FONT_16X12:ARRAY[0..255,0..31]OF BYTE :=[
16#00,16#00,16#00,16#00,16#00,16#00,16#00,16#00,16#00,16#00,16#00,16#00,16#00,16#00,16#00,16#00,16#00,16#00,16#00,16#00,16#00,16#00,16#00,16#00,16#00,16#00,16#00,16#00,16#00,16#00,16#00,16#00,	// 16#00
16#80,16#3F,16#80,16#3F,16#C0,16#60,16#C0,16#60,16#40,16#4A,16#40,16#4A,16#40,16#43,16#40,16#43,16#40,16#43,16#40,16#43,16#40,16#4A,16#40,16#4A,16#C0,16#60,16#C0,16#60,16#80,16#3F,16#80,16#3F,	// 16#01
16#80,16#3F,16#80,16#3F,16#C0,16#7F,16#C0,16#7F,16#C0,16#75,16#C0,16#75,16#C0,16#7C,16#C0,16#7C,16#C0,16#7C,16#C0,16#7C,16#C0,16#75,16#C0,16#75,16#C0,16#7F,16#C0,16#7F,16#80,16#3F,16#80,16#3F,	// 16#02
16#00,16#0E,16#00,16#1E,16#00,16#3F,16#00,16#3F,16#80,16#3F,16#80,16#1F,16#C0,16#0F,16#C0,16#0F,16#80,16#1F,16#80,16#3F,16#00,16#3F,16#00,16#3F,16#00,16#1E,16#00,16#0E,16#00,16#00,16#00,16#00,	// 16#03
16#00,16#0C,16#00,16#0C,16#00,16#1E,16#00,16#1E,16#00,16#3F,16#00,16#3F,16#80,16#7F,16#80,16#7F,16#00,16#3F,16#00,16#3F,16#00,16#1E,16#00,16#1E,16#00,16#0C,16#00,16#0C,16#00,16#00,16#00,16#00,	// 16#04
16#00,16#0E,16#00,16#0E,16#40,16#0E,16#40,16#0E,16#40,16#3E,16#40,16#3E,16#C0,16#79,16#C0,16#79,16#C0,16#79,16#C0,16#79,16#40,16#3E,16#40,16#3E,16#40,16#0E,16#40,16#0E,16#00,16#0E,16#00,16#0E,	// 16#05
16#00,16#0C,16#00,16#0C,16#40,16#1E,16#40,16#1E,16#40,16#3E,16#40,16#3E,16#C0,16#7F,16#C0,16#7F,16#C0,16#7F,16#C0,16#7F,16#40,16#3E,16#40,16#3E,16#40,16#1E,16#40,16#1E,16#00,16#0C,16#00,16#0C,	// 16#06
16#00,16#00,16#00,16#00,16#00,16#00,16#00,16#00,16#00,16#00,16#00,16#00,16#00,16#00,16#00,16#00,16#00,16#00,16#00,16#00,16#00,16#00,16#00,16#00,16#00,16#00,16#00,16#00,16#00,16#00,16#00,16#00,	// 16#07
16#00,16#00,16#00,16#00,16#00,16#00,16#00,16#00,16#00,16#00,16#00,16#00,16#00,16#00,16#00,16#00,16#00,16#00,16#00,16#00,16#00,16#00,16#00,16#00,16#00,16#00,16#00,16#00,16#00,16#00,16#00,16#00,	// 16#08
16#00,16#00,16#00,16#00,16#00,16#00,16#00,16#00,16#00,16#00,16#00,16#00,16#00,16#00,16#00,16#00,16#00,16#00,16#00,16#00,16#00,16#00,16#00,16#00,16#00,16#00,16#00,16#00,16#00,16#00,16#00,16#00,	// 16#09
16#00,16#00,16#00,16#00,16#00,16#00,16#00,16#00,16#00,16#00,16#00,16#00,16#00,16#00,16#00,16#00,16#00,16#00,16#00,16#00,16#00,16#00,16#00,16#00,16#00,16#00,16#00,16#00,16#00,16#00,16#00,16#00,	// 16#0A
16#80,16#07,16#80,16#07,16#C0,16#0F,16#C0,16#0F,16#40,16#4C,16#40,16#4C,16#40,16#5C,16#40,16#5C,16#C0,16#77,16#C0,16#77,16#80,16#63,16#80,16#63,16#00,16#78,16#00,16#78,16#00,16#00,16#00,16#00,	// 16#0B
16#00,16#00,16#00,16#00,16#00,16#39,16#00,16#39,16#00,16#7D,16#00,16#7D,16#C0,16#47,16#C0,16#47,16#C0,16#47,16#C0,16#47,16#00,16#7D,16#00,16#7D,16#00,16#39,16#00,16#39,16#00,16#00,16#00,16#00,	// 16#0C
16#00,16#00,16#00,16#00,16#00,16#00,16#00,16#00,16#00,16#00,16#00,16#00,16#00,16#00,16#00,16#00,16#00,16#00,16#00,16#00,16#00,16#00,16#00,16#00,16#00,16#00,16#00,16#00,16#00,16#00,16#00,16#00,	// 16#0D
16#C0,16#00,16#E0,16#00,16#E0,16#7F,16#E0,16#7F,16#C0,16#7F,16#80,16#7F,16#00,16#50,16#00,16#50,16#00,16#50,16#00,16#50,16#80,16#51,16#C0,16#51,16#C0,16#7F,16#C0,16#7F,16#80,16#7F,16#00,16#7F,	// 16#0E
16#80,16#16,16#80,16#16,16#80,16#1F,16#80,16#1F,16#00,16#0F,16#00,16#0F,16#C0,16#39,16#C0,16#39,16#C0,16#39,16#C0,16#39,16#00,16#0F,16#00,16#0F,16#80,16#1F,16#80,16#1F,16#80,16#16,16#80,16#16,	// 16#0F
16#C0,16#7F,16#C0,16#7F,16#80,16#3F,16#80,16#3F,16#00,16#1F,16#00,16#1F,16#00,16#0E,16#00,16#0E,16#00,16#0E,16#00,16#0E,16#00,16#04,16#00,16#04,16#00,16#04,16#00,16#04,16#00,16#00,16#00,16#00,	// 16#10
16#00,16#04,16#00,16#04,16#00,16#04,16#00,16#04,16#00,16#0E,16#00,16#0E,16#00,16#0E,16#00,16#0E,16#00,16#1F,16#00,16#1F,16#80,16#3F,16#80,16#3F,16#C0,16#7F,16#C0,16#7F,16#00,16#00,16#00,16#00,	// 16#11
16#00,16#00,16#00,16#00,16#00,16#11,16#00,16#11,16#80,16#31,16#80,16#31,16#C0,16#7F,16#C0,16#7F,16#C0,16#7F,16#C0,16#7F,16#80,16#31,16#80,16#31,16#00,16#11,16#00,16#11,16#00,16#00,16#00,16#00,	// 16#12
16#00,16#00,16#00,16#00,16#C0,16#7C,16#C0,16#7C,16#C0,16#7C,16#C0,16#7C,16#00,16#00,16#00,16#00,16#00,16#00,16#00,16#00,16#C0,16#7C,16#C0,16#7C,16#C0,16#7C,16#C0,16#7C,16#00,16#00,16#00,16#00,	// 16#13
16#00,16#38,16#00,16#38,16#00,16#7C,16#00,16#7C,16#00,16#44,16#00,16#44,16#C0,16#7F,16#C0,16#7F,16#C0,16#7F,16#C0,16#7F,16#00,16#40,16#00,16#40,16#C0,16#7F,16#C0,16#7F,16#C0,16#7F,16#C0,16#7F,	// 16#14
16#40,16#00,16#40,16#00,16#60,16#26,16#60,16#36,16#20,16#7F,16#20,16#7F,16#20,16#59,16#20,16#49,16#20,16#49,16#A0,16#49,16#E0,16#4F,16#E0,16#4F,16#C0,16#66,16#40,16#66,16#00,16#20,16#00,16#20,	// 16#15
16#C0,16#01,16#C0,16#01,16#C0,16#01,16#C0,16#01,16#C0,16#01,16#C0,16#01,16#C0,16#01,16#C0,16#01,16#C0,16#01,16#C0,16#01,16#C0,16#01,16#C0,16#01,16#C0,16#01,16#C0,16#01,16#00,16#00,16#00,16#00,	// 16#16
16#00,16#00,16#00,16#00,16#20,16#11,16#20,16#11,16#A0,16#31,16#A0,16#31,16#E0,16#7F,16#E0,16#7F,16#E0,16#7F,16#E0,16#7F,16#A0,16#31,16#A0,16#31,16#20,16#11,16#20,16#11,16#00,16#00,16#00,16#00,	// 16#17
16#00,16#00,16#00,16#00,16#00,16#10,16#00,16#10,16#00,16#30,16#00,16#30,16#C0,16#7F,16#C0,16#7F,16#C0,16#7F,16#C0,16#7F,16#00,16#30,16#00,16#30,16#00,16#10,16#00,16#10,16#00,16#00,16#00,16#00,	// 16#18
16#00,16#00,16#00,16#00,16#00,16#01,16#00,16#01,16#80,16#01,16#80,16#01,16#C0,16#7F,16#C0,16#7F,16#C0,16#7F,16#C0,16#7F,16#80,16#01,16#80,16#01,16#00,16#01,16#00,16#01,16#00,16#00,16#00,16#00,	// 16#19
16#00,16#04,16#00,16#04,16#00,16#04,16#00,16#04,16#00,16#04,16#00,16#04,16#00,16#15,16#00,16#15,16#00,16#1F,16#00,16#1F,16#00,16#0E,16#00,16#0E,16#00,16#04,16#00,16#04,16#00,16#00,16#00,16#00,	// 16#1A
16#00,16#04,16#00,16#04,16#00,16#0E,16#00,16#0E,16#00,16#1F,16#00,16#1F,16#00,16#15,16#00,16#15,16#00,16#04,16#00,16#04,16#00,16#04,16#00,16#04,16#00,16#04,16#00,16#04,16#00,16#00,16#00,16#00,	// 16#1B
16#00,16#0F,16#00,16#0F,16#00,16#0F,16#00,16#0F,16#00,16#01,16#00,16#01,16#00,16#01,16#00,16#01,16#00,16#01,16#00,16#01,16#00,16#01,16#00,16#01,16#00,16#01,16#00,16#01,16#00,16#00,16#00,16#00,	// 16#1C
16#00,16#04,16#00,16#04,16#00,16#0E,16#00,16#0E,16#00,16#1F,16#00,16#1F,16#00,16#04,16#00,16#04,16#00,16#04,16#00,16#04,16#00,16#1F,16#00,16#1F,16#00,16#0E,16#00,16#0E,16#00,16#04,16#00,16#04,	// 16#1D
16#C0,16#00,16#C0,16#01,16#C0,16#03,16#C0,16#07,16#C0,16#0F,16#C0,16#1F,16#C0,16#3F,16#C0,16#3F,16#C0,16#1F,16#C0,16#0F,16#C0,16#07,16#C0,16#03,16#C0,16#01,16#C0,16#00,16#00,16#00,16#00,16#00,	// 16#1E
16#00,16#30,16#00,16#38,16#00,16#3C,16#00,16#3E,16#00,16#3F,16#80,16#3F,16#C0,16#3F,16#C0,16#3F,16#80,16#3F,16#00,16#3F,16#00,16#3E,16#00,16#3C,16#00,16#38,16#00,16#30,16#00,16#00,16#00,16#00,	// 16#1F
16#00,16#00,16#00,16#00,16#00,16#00,16#00,16#00,16#00,16#00,16#00,16#00,16#00,16#00,16#00,16#00,16#00,16#00,16#00,16#00,16#00,16#00,16#00,16#00,16#00,16#00,16#00,16#00,16#00,16#00,16#00,16#00,	// 16#20
16#00,16#00,16#00,16#00,16#00,16#10,16#00,16#38,16#C0,16#7E,16#C0,16#7E,16#C0,16#7E,16#C0,16#7E,16#00,16#38,16#00,16#10,16#00,16#00,16#00,16#00,16#00,16#00,16#00,16#00,16#00,16#00,16#00,16#00,	// 16#21
16#00,16#00,16#00,16#00,16#00,16#60,16#00,16#70,16#00,16#78,16#00,16#78,16#00,16#00,16#00,16#00,16#00,16#00,16#00,16#00,16#00,16#78,16#00,16#78,16#00,16#70,16#00,16#60,16#00,16#00,16#00,16#00,	// 16#22
16#00,16#11,16#00,16#11,16#C0,16#7F,16#C0,16#7F,16#C0,16#7F,16#C0,16#7F,16#00,16#11,16#00,16#11,16#C0,16#7F,16#C0,16#7F,16#C0,16#7F,16#C0,16#7F,16#00,16#11,16#00,16#11,16#00,16#00,16#00,16#00,	// 16#23
16#80,16#18,16#80,16#18,16#80,16#3C,16#80,16#3C,16#E0,16#E4,16#E0,16#E4,16#E0,16#E4,16#E0,16#E4,16#80,16#27,16#80,16#27,16#00,16#23,16#00,16#23,16#00,16#00,16#00,16#00,16#00,16#00,16#00,16#00,	// 16#24
16#C0,16#18,16#C0,16#18,16#80,16#19,16#80,16#19,16#00,16#03,16#00,16#03,16#00,16#06,16#00,16#06,16#C0,16#0C,16#C0,16#0C,16#C0,16#18,16#C0,16#18,16#00,16#00,16#00,16#00,16#00,16#00,16#00,16#00,	// 16#25
16#80,16#37,16#80,16#37,16#C0,16#7F,16#C0,16#7F,16#40,16#4C,16#40,16#4C,16#C0,16#7C,16#C0,16#7E,16#80,16#37,16#80,16#37,16#C0,16#03,16#C0,16#02,16#40,16#06,16#40,16#06,16#00,16#00,16#00,16#00,	// 16#26
16#00,16#00,16#00,16#00,16#00,16#08,16#00,16#08,16#00,16#78,16#00,16#78,16#00,16#70,16#00,16#60,16#00,16#00,16#00,16#00,16#00,16#00,16#00,16#00,16#00,16#00,16#00,16#00,16#00,16#00,16#00,16#00,	// 16#27
16#00,16#00,16#00,16#00,16#00,16#1F,16#00,16#1F,16#80,16#3F,16#80,16#3F,16#C0,16#60,16#C0,16#60,16#40,16#40,16#40,16#40,16#00,16#00,16#00,16#00,16#00,16#00,16#00,16#00,16#00,16#00,16#00,16#00,	// 16#28
16#00,16#00,16#00,16#00,16#00,16#00,16#00,16#00,16#40,16#40,16#40,16#40,16#C0,16#60,16#C0,16#60,16#80,16#3F,16#80,16#3F,16#00,16#1F,16#00,16#1F,16#00,16#00,16#00,16#00,16#00,16#00,16#00,16#00,	// 16#29
16#00,16#04,16#00,16#04,16#00,16#15,16#00,16#15,16#00,16#1F,16#00,16#1F,16#00,16#0E,16#00,16#0E,16#00,16#0E,16#00,16#0E,16#00,16#1F,16#00,16#1F,16#00,16#15,16#00,16#15,16#00,16#04,16#00,16#04,	// 16#2A
16#00,16#00,16#00,16#00,16#00,16#04,16#00,16#04,16#00,16#04,16#00,16#04,16#00,16#1F,16#00,16#1F,16#00,16#1F,16#00,16#1F,16#00,16#04,16#00,16#04,16#00,16#04,16#00,16#04,16#00,16#00,16#00,16#00,	// 16#2B
16#00,16#00,16#00,16#00,16#20,16#00,16#20,16#00,16#E0,16#00,16#E0,16#00,16#C0,16#00,16#C0,16#00,16#C0,16#00,16#80,16#00,16#00,16#00,16#00,16#00,16#00,16#00,16#00,16#00,16#00,16#00,16#00,16#00,	// 16#2C
16#00,16#04,16#00,16#04,16#00,16#04,16#00,16#04,16#00,16#04,16#00,16#04,16#00,16#04,16#00,16#04,16#00,16#04,16#00,16#04,16#00,16#04,16#00,16#04,16#00,16#04,16#00,16#04,16#00,16#00,16#00,16#00,	// 16#2D
16#00,16#00,16#00,16#00,16#00,16#00,16#00,16#00,16#C0,16#00,16#C0,16#00,16#C0,16#00,16#C0,16#00,16#C0,16#00,16#C0,16#00,16#00,16#00,16#00,16#00,16#00,16#00,16#00,16#00,16#00,16#00,16#00,16#00,	// 16#2E
16#C0,16#00,16#C0,16#00,16#80,16#01,16#80,16#01,16#00,16#03,16#00,16#03,16#00,16#06,16#00,16#06,16#00,16#0C,16#00,16#0C,16#00,16#18,16#00,16#18,16#00,16#30,16#00,16#30,16#00,16#00,16#00,16#00,	// 16#2F
16#80,16#3F,16#80,16#3F,16#C0,16#7F,16#C0,16#7F,16#C0,16#41,16#40,16#43,16#40,16#46,16#40,16#4C,16#40,16#58,16#40,16#70,16#C0,16#7F,16#C0,16#7F,16#80,16#3F,16#80,16#3F,16#00,16#00,16#00,16#00,	// 16#30
16#40,16#10,16#40,16#10,16#40,16#10,16#40,16#10,16#C0,16#3F,16#C0,16#3F,16#C0,16#7F,16#C0,16#7F,16#40,16#00,16#40,16#00,16#40,16#00,16#40,16#00,16#00,16#00,16#00,16#00,16#00,16#00,16#00,16#00,	// 16#31
16#C0,16#30,16#C0,16#30,16#C0,16#71,16#C0,16#71,16#40,16#43,16#40,16#43,16#40,16#46,16#40,16#46,16#C0,16#7C,16#C0,16#7C,16#C0,16#38,16#C0,16#38,16#00,16#00,16#00,16#00,16#00,16#00,16#00,16#00,	// 16#32
16#80,16#20,16#80,16#20,16#C0,16#60,16#C0,16#60,16#40,16#44,16#40,16#44,16#40,16#44,16#40,16#44,16#C0,16#7F,16#C0,16#7F,16#80,16#3B,16#80,16#3B,16#00,16#00,16#00,16#00,16#00,16#00,16#00,16#00,	// 16#33
16#00,16#06,16#00,16#06,16#00,16#0E,16#00,16#0E,16#00,16#1A,16#00,16#1A,16#40,16#32,16#40,16#32,16#C0,16#7F,16#C0,16#7F,16#C0,16#7F,16#C0,16#7F,16#40,16#02,16#40,16#02,16#00,16#00,16#00,16#00,	// 16#34
16#80,16#7C,16#80,16#7C,16#C0,16#7C,16#C0,16#7C,16#40,16#44,16#40,16#44,16#40,16#44,16#40,16#44,16#C0,16#47,16#C0,16#47,16#80,16#43,16#80,16#43,16#00,16#00,16#00,16#00,16#00,16#00,16#00,16#00,	// 16#35
16#80,16#1F,16#80,16#1F,16#C0,16#3F,16#C0,16#3F,16#40,16#64,16#40,16#64,16#40,16#44,16#40,16#44,16#C0,16#47,16#C0,16#47,16#80,16#03,16#80,16#03,16#00,16#00,16#00,16#00,16#00,16#00,16#00,16#00,	// 16#36
16#00,16#70,16#00,16#70,16#00,16#70,16#00,16#70,16#C0,16#41,16#C0,16#41,16#C0,16#43,16#C0,16#43,16#00,16#46,16#00,16#46,16#00,16#7C,16#00,16#7C,16#00,16#78,16#00,16#78,16#00,16#00,16#00,16#00,	// 16#37
16#80,16#3B,16#80,16#3B,16#C0,16#7F,16#C0,16#7F,16#40,16#44,16#40,16#44,16#40,16#44,16#40,16#44,16#C0,16#7F,16#C0,16#7F,16#80,16#3B,16#80,16#3B,16#00,16#00,16#00,16#00,16#00,16#00,16#00,16#00,	// 16#38
16#00,16#38,16#00,16#38,16#40,16#7C,16#40,16#7C,16#C0,16#44,16#C0,16#44,16#C0,16#47,16#C0,16#47,16#00,16#7F,16#00,16#7F,16#00,16#3C,16#00,16#3C,16#00,16#00,16#00,16#00,16#00,16#00,16#00,16#00,	// 16#39
16#00,16#00,16#00,16#00,16#00,16#00,16#00,16#00,16#80,16#19,16#80,16#19,16#80,16#19,16#80,16#19,16#80,16#19,16#80,16#19,16#00,16#00,16#00,16#00,16#00,16#00,16#00,16#00,16#00,16#00,16#00,16#00,	// 16#3A
16#00,16#00,16#00,16#00,16#00,16#00,16#00,16#00,16#A0,16#19,16#A0,16#19,16#E0,16#19,16#E0,16#19,16#C0,16#19,16#C0,16#19,16#00,16#00,16#00,16#00,16#00,16#00,16#00,16#00,16#00,16#00,16#00,16#00,	// 16#3B
16#00,16#04,16#00,16#04,16#00,16#0E,16#00,16#0E,16#00,16#1B,16#00,16#1B,16#80,16#31,16#80,16#31,16#C0,16#60,16#C0,16#60,16#40,16#40,16#40,16#40,16#00,16#00,16#00,16#00,16#00,16#00,16#00,16#00,	// 16#3C
16#00,16#00,16#00,16#00,16#00,16#0A,16#00,16#0A,16#00,16#0A,16#00,16#0A,16#00,16#0A,16#00,16#0A,16#00,16#0A,16#00,16#0A,16#00,16#0A,16#00,16#0A,16#00,16#0A,16#00,16#0A,16#00,16#00,16#00,16#00,	// 16#3D
16#00,16#00,16#00,16#00,16#40,16#40,16#40,16#40,16#C0,16#60,16#C0,16#60,16#80,16#31,16#80,16#31,16#00,16#1B,16#00,16#1B,16#00,16#0E,16#00,16#0E,16#00,16#04,16#00,16#04,16#00,16#00,16#00,16#00,	// 16#3E
16#00,16#20,16#00,16#20,16#00,16#60,16#00,16#60,16#C0,16#46,16#C0,16#46,16#C0,16#4E,16#C0,16#4E,16#00,16#78,16#00,16#78,16#00,16#30,16#00,16#30,16#00,16#00,16#00,16#00,16#00,16#00,16#00,16#00,	// 16#3F
16#80,16#3F,16#80,16#3F,16#C0,16#7F,16#C0,16#7F,16#40,16#40,16#40,16#40,16#40,16#4E,16#40,16#4E,16#40,16#4A,16#40,16#4A,16#40,16#7A,16#40,16#7E,16#00,16#3E,16#00,16#3E,16#00,16#00,16#00,16#00,	// 16#40
16#C0,16#1F,16#C0,16#1F,16#C0,16#3F,16#C0,16#3F,16#00,16#62,16#00,16#62,16#00,16#62,16#00,16#62,16#C0,16#3F,16#C0,16#3F,16#C0,16#1F,16#C0,16#1F,16#00,16#00,16#00,16#00,16#00,16#00,16#00,16#00,	// 16#41
16#40,16#40,16#40,16#40,16#C0,16#7F,16#C0,16#7F,16#C0,16#7F,16#C0,16#7F,16#40,16#44,16#40,16#44,16#40,16#44,16#40,16#44,16#C0,16#7F,16#C0,16#7F,16#80,16#3B,16#80,16#3B,16#00,16#00,16#00,16#00,	// 16#42
16#00,16#1F,16#00,16#1F,16#80,16#3F,16#80,16#3F,16#C0,16#60,16#C0,16#60,16#40,16#40,16#40,16#40,16#40,16#40,16#40,16#40,16#C0,16#71,16#C0,16#71,16#80,16#31,16#80,16#31,16#00,16#00,16#00,16#00,	// 16#43
16#40,16#40,16#40,16#40,16#C0,16#7F,16#C0,16#7F,16#C0,16#7F,16#C0,16#7F,16#40,16#40,16#40,16#40,16#C0,16#60,16#C0,16#60,16#80,16#3F,16#80,16#3F,16#00,16#1F,16#00,16#1F,16#00,16#00,16#00,16#00,	// 16#44
16#40,16#40,16#40,16#40,16#C0,16#7F,16#C0,16#7F,16#C0,16#7F,16#C0,16#7F,16#40,16#44,16#40,16#44,16#40,16#44,16#40,16#44,16#40,16#4E,16#40,16#4E,16#C0,16#60,16#C0,16#60,16#00,16#00,16#00,16#00,	// 16#45
16#40,16#40,16#40,16#40,16#C0,16#7F,16#C0,16#7F,16#C0,16#7F,16#C0,16#7F,16#40,16#44,16#40,16#44,16#00,16#44,16#00,16#44,16#00,16#6E,16#00,16#6E,16#00,16#70,16#00,16#70,16#00,16#00,16#00,16#00,	// 16#46
16#00,16#1F,16#00,16#1F,16#80,16#3F,16#80,16#3F,16#C0,16#60,16#C0,16#60,16#40,16#40,16#40,16#40,16#40,16#42,16#40,16#42,16#C0,16#73,16#C0,16#73,16#C0,16#33,16#C0,16#33,16#00,16#00,16#00,16#00,	// 16#47
16#C0,16#7F,16#C0,16#7F,16#C0,16#7F,16#C0,16#7F,16#00,16#04,16#00,16#04,16#00,16#04,16#00,16#04,16#C0,16#7F,16#C0,16#7F,16#C0,16#7F,16#C0,16#7F,16#00,16#00,16#00,16#00,16#00,16#00,16#00,16#00,	// 16#48
16#00,16#00,16#00,16#00,16#40,16#40,16#40,16#40,16#C0,16#7F,16#C0,16#7F,16#C0,16#7F,16#C0,16#7F,16#40,16#40,16#40,16#40,16#00,16#00,16#00,16#00,16#00,16#00,16#00,16#00,16#00,16#00,16#00,16#00,	// 16#49
16#80,16#03,16#80,16#03,16#C0,16#03,16#C0,16#03,16#40,16#00,16#40,16#00,16#40,16#40,16#40,16#40,16#C0,16#7F,16#C0,16#7F,16#80,16#7F,16#80,16#7F,16#00,16#40,16#00,16#40,16#00,16#00,16#00,16#00,	// 16#4A
16#40,16#40,16#40,16#40,16#C0,16#7F,16#C0,16#7F,16#C0,16#7F,16#C0,16#7F,16#00,16#04,16#00,16#04,16#00,16#0E,16#00,16#1F,16#C0,16#7B,16#C0,16#71,16#C0,16#60,16#C0,16#60,16#00,16#00,16#00,16#00,	// 16#4B
16#40,16#40,16#40,16#40,16#C0,16#7F,16#C0,16#7F,16#C0,16#7F,16#C0,16#7F,16#40,16#40,16#40,16#40,16#40,16#00,16#40,16#00,16#C0,16#01,16#C0,16#01,16#C0,16#03,16#C0,16#03,16#00,16#00,16#00,16#00,	// 16#4C
16#C0,16#7F,16#C0,16#7F,16#C0,16#7F,16#C0,16#7F,16#00,16#38,16#00,16#38,16#00,16#1C,16#00,16#1C,16#00,16#38,16#00,16#38,16#C0,16#7F,16#C0,16#7F,16#C0,16#7F,16#C0,16#7F,16#00,16#00,16#00,16#00,	// 16#4D
16#C0,16#7F,16#C0,16#7F,16#C0,16#7F,16#C0,16#7F,16#00,16#1C,16#00,16#1C,16#00,16#0E,16#00,16#0E,16#00,16#07,16#00,16#07,16#C0,16#7F,16#C0,16#7F,16#C0,16#7F,16#C0,16#7F,16#00,16#00,16#00,16#00,	// 16#4E
16#00,16#1F,16#00,16#1F,16#80,16#3F,16#80,16#3F,16#C0,16#71,16#C0,16#60,16#40,16#40,16#40,16#40,16#C0,16#60,16#C0,16#71,16#80,16#3F,16#80,16#3F,16#00,16#1F,16#00,16#1F,16#00,16#00,16#00,16#00,	// 16#4F
16#40,16#40,16#40,16#40,16#C0,16#7F,16#C0,16#7F,16#C0,16#7F,16#C0,16#7F,16#40,16#44,16#40,16#44,16#00,16#44,16#00,16#44,16#00,16#7C,16#00,16#7C,16#00,16#38,16#00,16#38,16#00,16#00,16#00,16#00,	// 16#50
16#00,16#1F,16#00,16#1F,16#80,16#3F,16#80,16#3F,16#80,16#60,16#80,16#60,16#A0,16#40,16#A0,16#43,16#E0,16#63,16#E0,16#61,16#E0,16#3F,16#E0,16#3F,16#20,16#1F,16#20,16#1F,16#00,16#00,16#00,16#00,	// 16#51
16#40,16#40,16#40,16#40,16#C0,16#7F,16#C0,16#7F,16#C0,16#7F,16#C0,16#7F,16#00,16#44,16#00,16#44,16#00,16#46,16#00,16#46,16#C0,16#7F,16#C0,16#7F,16#C0,16#39,16#C0,16#39,16#00,16#00,16#00,16#00,	// 16#52
16#80,16#39,16#80,16#39,16#C0,16#7D,16#C0,16#7D,16#40,16#44,16#40,16#44,16#40,16#46,16#40,16#46,16#C0,16#73,16#C0,16#73,16#80,16#31,16#80,16#31,16#00,16#00,16#00,16#00,16#00,16#00,16#00,16#00,	// 16#53
16#00,16#60,16#00,16#60,16#40,16#40,16#40,16#40,16#C0,16#7F,16#C0,16#7F,16#C0,16#7F,16#C0,16#7F,16#40,16#40,16#40,16#40,16#00,16#60,16#00,16#60,16#00,16#00,16#00,16#00,16#00,16#00,16#00,16#00,	// 16#54
16#80,16#7F,16#80,16#7F,16#C0,16#7F,16#C0,16#7F,16#40,16#00,16#40,16#00,16#40,16#00,16#40,16#00,16#C0,16#7F,16#C0,16#7F,16#80,16#7F,16#80,16#7F,16#00,16#00,16#00,16#00,16#00,16#00,16#00,16#00,	// 16#55
16#00,16#7F,16#00,16#7F,16#80,16#7F,16#80,16#7F,16#C0,16#00,16#C0,16#00,16#C0,16#00,16#C0,16#00,16#80,16#7F,16#80,16#7F,16#00,16#7F,16#00,16#7F,16#00,16#00,16#00,16#00,16#00,16#00,16#00,16#00,	// 16#56
16#00,16#7E,16#00,16#7F,16#C0,16#7F,16#C0,16#7F,16#C0,16#01,16#C0,16#03,16#00,16#07,16#00,16#07,16#C0,16#03,16#C0,16#01,16#C0,16#7F,16#C0,16#7F,16#00,16#7F,16#00,16#7E,16#00,16#00,16#00,16#00,	// 16#57
16#C0,16#71,16#C0,16#71,16#C0,16#7B,16#C0,16#7B,16#00,16#0E,16#00,16#0E,16#00,16#0E,16#00,16#0E,16#C0,16#7B,16#C0,16#7B,16#C0,16#71,16#C0,16#71,16#00,16#00,16#00,16#00,16#00,16#00,16#00,16#00,	// 16#58
16#00,16#78,16#00,16#78,16#40,16#7C,16#40,16#7C,16#C0,16#07,16#C0,16#07,16#C0,16#07,16#C0,16#07,16#40,16#7C,16#40,16#7C,16#00,16#78,16#00,16#78,16#00,16#00,16#00,16#00,16#00,16#00,16#00,16#00,	// 16#59
16#C0,16#70,16#C0,16#71,16#C0,16#61,16#C0,16#63,16#40,16#47,16#40,16#46,16#40,16#4C,16#40,16#5C,16#40,16#58,16#40,16#58,16#C0,16#70,16#C0,16#70,16#C0,16#61,16#C0,16#61,16#00,16#00,16#00,16#00,	// 16#5A
16#00,16#00,16#00,16#00,16#00,16#00,16#00,16#00,16#C0,16#7F,16#C0,16#7F,16#C0,16#7F,16#C0,16#7F,16#40,16#40,16#40,16#40,16#40,16#40,16#40,16#40,16#00,16#00,16#00,16#00,16#00,16#00,16#00,16#00,	// 16#5B
16#00,16#30,16#00,16#30,16#00,16#18,16#00,16#18,16#00,16#0C,16#00,16#0C,16#00,16#06,16#00,16#06,16#00,16#03,16#00,16#03,16#80,16#01,16#80,16#01,16#C0,16#00,16#C0,16#00,16#00,16#00,16#00,16#00,	// 16#5C
16#00,16#00,16#00,16#00,16#00,16#00,16#00,16#00,16#40,16#40,16#40,16#40,16#40,16#40,16#40,16#40,16#C0,16#7F,16#C0,16#7F,16#C0,16#7F,16#C0,16#7F,16#00,16#00,16#00,16#00,16#00,16#00,16#00,16#00,	// 16#5D
16#00,16#10,16#00,16#10,16#00,16#30,16#00,16#30,16#00,16#60,16#00,16#60,16#00,16#C0,16#00,16#C0,16#00,16#60,16#00,16#60,16#00,16#30,16#00,16#30,16#00,16#10,16#00,16#10,16#00,16#00,16#00,16#00,	// 16#5E
16#20,16#00,16#20,16#00,16#20,16#00,16#20,16#00,16#20,16#00,16#20,16#00,16#20,16#00,16#20,16#00,16#20,16#00,16#20,16#00,16#20,16#00,16#20,16#00,16#20,16#00,16#20,16#00,16#20,16#00,16#20,16#00,	// 16#5F
16#00,16#00,16#00,16#00,16#00,16#00,16#00,16#00,16#00,16#C0,16#00,16#C0,16#00,16#E0,16#00,16#E0,16#00,16#20,16#00,16#20,16#00,16#00,16#00,16#00,16#00,16#00,16#00,16#00,16#00,16#00,16#00,16#00,	// 16#60
16#80,16#01,16#80,16#01,16#C0,16#0B,16#C0,16#0B,16#40,16#0A,16#40,16#0A,16#40,16#0A,16#40,16#0A,16#C0,16#0F,16#80,16#0F,16#80,16#07,16#C0,16#07,16#40,16#00,16#40,16#00,16#00,16#00,16#00,16#00,	// 16#61
16#40,16#40,16#40,16#40,16#C0,16#7F,16#80,16#7F,16#80,16#7F,16#C0,16#7F,16#40,16#08,16#40,16#08,16#40,16#08,16#40,16#08,16#C0,16#0F,16#C0,16#0F,16#80,16#07,16#80,16#07,16#00,16#00,16#00,16#00,	// 16#62
16#80,16#07,16#80,16#07,16#C0,16#0F,16#C0,16#0F,16#40,16#08,16#40,16#08,16#40,16#08,16#40,16#08,16#C0,16#0C,16#C0,16#0C,16#80,16#04,16#80,16#04,16#00,16#00,16#00,16#00,16#00,16#00,16#00,16#00,	// 16#63
16#80,16#07,16#80,16#07,16#C0,16#0F,16#C0,16#0F,16#40,16#08,16#40,16#08,16#40,16#48,16#40,16#48,16#C0,16#7F,16#80,16#7F,16#80,16#7F,16#C0,16#7F,16#40,16#00,16#40,16#00,16#00,16#00,16#00,16#00,	// 16#64
16#80,16#07,16#80,16#07,16#C0,16#0F,16#C0,16#0F,16#40,16#0A,16#40,16#0A,16#40,16#0A,16#40,16#0A,16#C0,16#0E,16#C0,16#0E,16#80,16#06,16#80,16#06,16#00,16#00,16#00,16#00,16#00,16#00,16#00,16#00,	// 16#65
16#40,16#04,16#40,16#04,16#C0,16#3F,16#C0,16#3F,16#C0,16#7F,16#C0,16#7F,16#40,16#44,16#40,16#44,16#00,16#64,16#00,16#64,16#00,16#20,16#00,16#20,16#00,16#00,16#00,16#00,16#00,16#00,16#00,16#00,	// 16#66
16#20,16#07,16#20,16#07,16#B0,16#0F,16#B0,16#0F,16#90,16#08,16#90,16#08,16#90,16#08,16#90,16#08,16#F0,16#0F,16#F0,16#07,16#E0,16#07,16#E0,16#0F,16#00,16#08,16#00,16#08,16#00,16#00,16#00,16#00,	// 16#67
16#40,16#40,16#40,16#40,16#C0,16#7F,16#C0,16#7F,16#C0,16#7F,16#C0,16#7F,16#00,16#04,16#00,16#04,16#00,16#08,16#00,16#08,16#C0,16#0F,16#C0,16#0F,16#C0,16#07,16#C0,16#07,16#00,16#00,16#00,16#00,	// 16#68
16#00,16#00,16#00,16#00,16#40,16#08,16#40,16#08,16#40,16#08,16#40,16#08,16#C0,16#6F,16#C0,16#6F,16#C0,16#6F,16#C0,16#6F,16#40,16#00,16#40,16#00,16#40,16#00,16#40,16#00,16#00,16#00,16#00,16#00,	// 16#69
16#60,16#00,16#60,16#00,16#70,16#00,16#70,16#00,16#10,16#08,16#10,16#08,16#10,16#08,16#10,16#08,16#F0,16#6F,16#F0,16#6F,16#E0,16#6F,16#E0,16#6F,16#00,16#00,16#00,16#00,16#00,16#00,16#00,16#00,	// 16#6A
16#40,16#40,16#40,16#40,16#C0,16#7F,16#C0,16#7F,16#C0,16#7F,16#C0,16#7F,16#00,16#02,16#00,16#02,16#00,16#07,16#00,16#07,16#C0,16#0D,16#C0,16#0D,16#C0,16#08,16#C0,16#08,16#00,16#00,16#00,16#00,	// 16#6B
16#00,16#00,16#00,16#00,16#40,16#40,16#40,16#40,16#40,16#40,16#40,16#40,16#C0,16#7F,16#C0,16#7F,16#C0,16#7F,16#C0,16#7F,16#40,16#00,16#40,16#00,16#40,16#00,16#40,16#00,16#00,16#00,16#00,16#00,	// 16#6C
16#C0,16#0F,16#C0,16#0F,16#C0,16#0F,16#C0,16#0F,16#00,16#08,16#00,16#08,16#80,16#0F,16#80,16#0F,16#00,16#08,16#00,16#08,16#C0,16#0F,16#C0,16#0F,16#C0,16#07,16#C0,16#07,16#00,16#00,16#00,16#00,	// 16#6D
16#C0,16#0F,16#C0,16#0F,16#C0,16#0F,16#C0,16#0F,16#00,16#08,16#00,16#08,16#00,16#08,16#00,16#08,16#C0,16#0F,16#C0,16#0F,16#C0,16#07,16#C0,16#07,16#00,16#00,16#00,16#00,16#00,16#00,16#00,16#00,	// 16#6E
16#80,16#07,16#80,16#07,16#C0,16#0F,16#C0,16#0F,16#40,16#08,16#40,16#08,16#40,16#08,16#40,16#08,16#C0,16#0F,16#C0,16#0F,16#80,16#07,16#80,16#07,16#00,16#00,16#00,16#00,16#00,16#00,16#00,16#00,	// 16#6F
16#10,16#08,16#10,16#08,16#F0,16#0F,16#F0,16#07,16#F0,16#07,16#F0,16#0F,16#50,16#08,16#50,16#08,16#40,16#08,16#40,16#08,16#C0,16#0F,16#C0,16#0F,16#80,16#07,16#80,16#07,16#00,16#00,16#00,16#00,	// 16#70
16#80,16#07,16#80,16#07,16#C0,16#0F,16#C0,16#0F,16#40,16#08,16#40,16#08,16#50,16#08,16#50,16#08,16#F0,16#0F,16#F0,16#07,16#F0,16#07,16#F0,16#0F,16#10,16#08,16#10,16#08,16#00,16#00,16#00,16#00,	// 16#71
16#40,16#08,16#40,16#08,16#C0,16#0F,16#C0,16#0F,16#C0,16#0F,16#C0,16#0F,16#40,16#02,16#40,16#06,16#00,16#0C,16#00,16#0C,16#00,16#0E,16#00,16#0E,16#00,16#06,16#00,16#06,16#00,16#00,16#00,16#00,	// 16#72
16#80,16#04,16#80,16#04,16#C0,16#0E,16#C0,16#0E,16#40,16#0A,16#40,16#0B,16#40,16#0B,16#40,16#09,16#C0,16#0D,16#C0,16#0D,16#80,16#04,16#80,16#04,16#00,16#00,16#00,16#00,16#00,16#00,16#00,16#00,	// 16#73
16#00,16#08,16#00,16#08,16#80,16#1F,16#80,16#1F,16#C0,16#3F,16#C0,16#3F,16#40,16#08,16#40,16#08,16#C0,16#08,16#C0,16#08,16#80,16#08,16#80,16#08,16#00,16#00,16#00,16#00,16#00,16#00,16#00,16#00,	// 16#74
16#80,16#0F,16#80,16#0F,16#C0,16#0F,16#C0,16#0F,16#40,16#00,16#40,16#00,16#40,16#00,16#40,16#00,16#80,16#0F,16#80,16#0F,16#C0,16#0F,16#C0,16#0F,16#40,16#00,16#40,16#00,16#00,16#00,16#00,16#00,	// 16#75
16#00,16#0F,16#00,16#0F,16#80,16#0F,16#80,16#0F,16#C0,16#00,16#C0,16#00,16#C0,16#00,16#C0,16#00,16#80,16#0F,16#80,16#0F,16#00,16#0F,16#00,16#0F,16#00,16#00,16#00,16#00,16#00,16#00,16#00,16#00,	// 16#76
16#00,16#0F,16#00,16#0F,16#C0,16#0F,16#C0,16#0F,16#C0,16#00,16#C0,16#00,16#00,16#03,16#00,16#03,16#C0,16#00,16#C0,16#00,16#C0,16#0F,16#C0,16#0F,16#00,16#0F,16#00,16#0F,16#00,16#00,16#00,16#00,	// 16#77
16#40,16#08,16#40,16#08,16#C0,16#0C,16#C0,16#0C,16#80,16#07,16#80,16#07,16#00,16#03,16#00,16#03,16#80,16#07,16#80,16#07,16#C0,16#0C,16#C0,16#0C,16#40,16#08,16#40,16#08,16#00,16#00,16#00,16#00,	// 16#78
16#10,16#00,16#10,16#00,16#10,16#0F,16#10,16#0F,16#90,16#0F,16#90,16#0F,16#B0,16#00,16#B0,16#00,16#E0,16#00,16#E0,16#00,16#C0,16#0F,16#C0,16#0F,16#00,16#0F,16#00,16#0F,16#00,16#00,16#00,16#00,	// 16#79
16#C0,16#0C,16#C0,16#0C,16#C0,16#09,16#C0,16#09,16#40,16#09,16#40,16#0B,16#40,16#0B,16#40,16#0A,16#40,16#0E,16#40,16#0E,16#C0,16#0C,16#C0,16#0C,16#00,16#00,16#00,16#00,16#00,16#00,16#00,16#00,	// 16#7A
16#00,16#04,16#00,16#04,16#00,16#0E,16#00,16#0E,16#80,16#3B,16#80,16#3B,16#C0,16#71,16#C0,16#71,16#40,16#40,16#40,16#40,16#40,16#40,16#40,16#40,16#00,16#00,16#00,16#00,16#00,16#00,16#00,16#00,	// 16#7B
16#00,16#00,16#00,16#00,16#00,16#00,16#00,16#00,16#00,16#00,16#00,16#00,16#C0,16#7B,16#C0,16#7B,16#C0,16#7B,16#C0,16#7B,16#00,16#00,16#00,16#00,16#00,16#00,16#00,16#00,16#00,16#00,16#00,16#00,	// 16#7C
16#40,16#40,16#40,16#40,16#40,16#40,16#40,16#40,16#C0,16#71,16#C0,16#71,16#80,16#3B,16#80,16#3B,16#00,16#0E,16#00,16#0E,16#00,16#04,16#00,16#04,16#00,16#00,16#00,16#00,16#00,16#00,16#00,16#00,	// 16#7D
16#00,16#30,16#00,16#30,16#00,16#70,16#00,16#60,16#00,16#40,16#00,16#40,16#00,16#60,16#00,16#60,16#00,16#30,16#00,16#30,16#00,16#10,16#00,16#10,16#00,16#30,16#00,16#70,16#00,16#60,16#00,16#40,	// 16#7E
16#80,16#03,16#80,16#03,16#80,16#07,16#80,16#07,16#80,16#0C,16#80,16#0C,16#80,16#18,16#80,16#18,16#80,16#0C,16#80,16#0C,16#80,16#07,16#80,16#07,16#80,16#03,16#80,16#03,16#00,16#00,16#00,16#00,	// 16#7F
16#80,16#3F,16#90,16#3F,16#D0,16#7F,16#D0,16#7F,16#70,16#40,16#70,16#40,16#70,16#40,16#60,16#40,16#C0,16#71,16#C0,16#71,16#80,16#31,16#80,16#31,16#00,16#00,16#00,16#00,16#00,16#00,16#00,16#00,	// 16#80
16#80,16#6F,16#80,16#6F,16#C0,16#6F,16#C0,16#6F,16#40,16#00,16#40,16#00,16#40,16#00,16#40,16#00,16#C0,16#6F,16#80,16#6F,16#80,16#6F,16#C0,16#6F,16#40,16#00,16#40,16#00,16#00,16#00,16#00,16#00,	// 16#81
16#80,16#07,16#80,16#07,16#C0,16#0F,16#C0,16#0F,16#40,16#2A,16#40,16#2A,16#40,16#6A,16#40,16#6A,16#C0,16#CE,16#C0,16#CE,16#80,16#86,16#80,16#86,16#00,16#00,16#00,16#00,16#00,16#00,16#00,16#00,	// 16#82
16#80,16#21,16#80,16#21,16#C0,16#6B,16#C0,16#6B,16#40,16#CA,16#40,16#CA,16#40,16#CA,16#40,16#CA,16#C0,16#6F,16#80,16#6F,16#80,16#27,16#C0,16#27,16#40,16#00,16#40,16#00,16#00,16#00,16#00,16#00,	// 16#83
16#80,16#61,16#80,16#61,16#C0,16#6B,16#C0,16#6B,16#40,16#0A,16#40,16#0A,16#40,16#0A,16#40,16#0A,16#C0,16#6F,16#80,16#6F,16#80,16#67,16#C0,16#67,16#40,16#00,16#40,16#00,16#00,16#00,16#00,16#00,	// 16#84
16#80,16#81,16#80,16#81,16#C0,16#CB,16#C0,16#CB,16#40,16#6A,16#40,16#6A,16#40,16#2A,16#40,16#2A,16#C0,16#0F,16#80,16#0F,16#80,16#07,16#C0,16#07,16#40,16#00,16#40,16#00,16#00,16#00,16#00,16#00,	// 16#85
16#80,16#09,16#80,16#09,16#C0,16#6B,16#C0,16#6B,16#40,16#FA,16#40,16#FA,16#40,16#9A,16#40,16#9A,16#C0,16#FF,16#80,16#FF,16#80,16#67,16#C0,16#67,16#40,16#00,16#40,16#00,16#00,16#00,16#00,16#00,	// 16#86
16#80,16#07,16#90,16#07,16#D0,16#0F,16#D0,16#0F,16#70,16#08,16#70,16#08,16#70,16#08,16#60,16#08,16#C0,16#0C,16#C0,16#0C,16#80,16#04,16#80,16#04,16#00,16#00,16#00,16#00,16#00,16#00,16#00,16#00,	// 16#87
16#80,16#27,16#80,16#27,16#C0,16#6F,16#C0,16#6F,16#40,16#CA,16#40,16#CA,16#40,16#CA,16#40,16#CA,16#40,16#6E,16#40,16#6E,16#40,16#26,16#40,16#26,16#00,16#00,16#00,16#00,16#00,16#00,16#00,16#00,	// 16#88
16#80,16#67,16#80,16#67,16#C0,16#6F,16#C0,16#6F,16#40,16#0A,16#40,16#0A,16#40,16#0A,16#40,16#0A,16#40,16#6E,16#40,16#6E,16#40,16#66,16#40,16#66,16#00,16#00,16#00,16#00,16#00,16#00,16#00,16#00,	// 16#89
16#80,16#87,16#80,16#87,16#C0,16#CF,16#C0,16#CF,16#40,16#6A,16#40,16#6A,16#40,16#2A,16#40,16#2A,16#40,16#0E,16#40,16#0E,16#40,16#06,16#40,16#06,16#00,16#00,16#00,16#00,16#00,16#00,16#00,16#00,	// 16#8A
16#00,16#00,16#00,16#00,16#40,16#68,16#40,16#68,16#40,16#68,16#40,16#68,16#C0,16#0F,16#C0,16#0F,16#C0,16#6F,16#C0,16#6F,16#40,16#60,16#40,16#60,16#40,16#00,16#40,16#00,16#00,16#00,16#00,16#00,	// 16#8B
16#00,16#00,16#00,16#00,16#40,16#28,16#40,16#28,16#40,16#68,16#40,16#68,16#C0,16#CF,16#C0,16#CF,16#C0,16#6F,16#C0,16#6F,16#40,16#20,16#40,16#20,16#40,16#00,16#40,16#00,16#00,16#00,16#00,16#00,	// 16#8C
16#00,16#00,16#00,16#00,16#40,16#88,16#40,16#88,16#40,16#C8,16#40,16#C8,16#C0,16#6F,16#C0,16#6F,16#C0,16#2F,16#C0,16#2F,16#40,16#00,16#40,16#00,16#40,16#00,16#40,16#00,16#00,16#00,16#00,16#00,	// 16#8D
16#C0,16#47,16#C0,16#47,16#C0,16#4F,16#C0,16#4F,16#00,16#19,16#00,16#19,16#00,16#19,16#00,16#19,16#C0,16#4F,16#C0,16#4F,16#C0,16#47,16#C0,16#47,16#00,16#00,16#00,16#00,16#00,16#00,16#00,16#00,	// 16#8E
16#C0,16#67,16#C0,16#67,16#C0,16#FF,16#C0,16#FF,16#00,16#99,16#00,16#99,16#00,16#99,16#00,16#99,16#C0,16#FF,16#C0,16#FF,16#C0,16#67,16#C0,16#67,16#00,16#00,16#00,16#00,16#00,16#00,16#00,16#00,	// 16#8F
16#C0,16#1F,16#C0,16#1F,16#C0,16#1F,16#C0,16#1F,16#40,16#32,16#40,16#32,16#40,16#72,16#40,16#72,16#40,16#D2,16#40,16#D2,16#C0,16#98,16#C0,16#98,16#00,16#00,16#00,16#00,16#00,16#00,16#00,16#00,	// 16#90
16#C0,16#01,16#C0,16#09,16#C0,16#0B,16#C0,16#0B,16#40,16#0A,16#40,16#0A,16#C0,16#0A,16#80,16#0F,16#80,16#0F,16#C0,16#0F,16#C0,16#0A,16#40,16#0A,16#40,16#0A,16#40,16#0E,16#40,16#06,16#40,16#06,	// 16#91
16#C0,16#1F,16#C0,16#1F,16#C0,16#3F,16#C0,16#3F,16#00,16#64,16#00,16#64,16#C0,16#7F,16#C0,16#7F,16#C0,16#7F,16#C0,16#7F,16#40,16#44,16#40,16#44,16#40,16#44,16#40,16#44,16#00,16#00,16#00,16#00,	// 16#92
16#80,16#27,16#80,16#27,16#C0,16#6F,16#C0,16#6F,16#40,16#C8,16#40,16#C8,16#40,16#C8,16#40,16#C8,16#C0,16#6F,16#C0,16#6F,16#80,16#27,16#80,16#27,16#00,16#00,16#00,16#00,16#00,16#00,16#00,16#00,	// 16#93
16#80,16#67,16#80,16#67,16#C0,16#6F,16#C0,16#6F,16#40,16#08,16#40,16#08,16#40,16#08,16#40,16#08,16#C0,16#6F,16#C0,16#6F,16#80,16#67,16#80,16#67,16#00,16#00,16#00,16#00,16#00,16#00,16#00,16#00,	// 16#94
16#80,16#87,16#80,16#87,16#C0,16#CF,16#C0,16#CF,16#40,16#68,16#40,16#68,16#40,16#28,16#40,16#28,16#C0,16#0F,16#C0,16#0F,16#80,16#07,16#80,16#07,16#00,16#00,16#00,16#00,16#00,16#00,16#00,16#00,	// 16#95
16#80,16#2F,16#80,16#2F,16#C0,16#6F,16#C0,16#6F,16#40,16#C0,16#40,16#C0,16#40,16#C0,16#40,16#C0,16#C0,16#6F,16#80,16#6F,16#80,16#2F,16#C0,16#2F,16#40,16#00,16#40,16#00,16#00,16#00,16#00,16#00,	// 16#96
16#80,16#8F,16#80,16#8F,16#C0,16#CF,16#C0,16#CF,16#40,16#60,16#40,16#60,16#40,16#20,16#40,16#20,16#C0,16#0F,16#80,16#0F,16#80,16#0F,16#C0,16#0F,16#40,16#00,16#40,16#00,16#00,16#00,16#00,16#00,	// 16#97
16#10,16#00,16#10,16#00,16#10,16#6F,16#10,16#6F,16#90,16#6F,16#90,16#6F,16#B0,16#00,16#B0,16#00,16#E0,16#00,16#E0,16#00,16#C0,16#6F,16#C0,16#6F,16#00,16#6F,16#00,16#6F,16#00,16#00,16#00,16#00,	// 16#98
16#80,16#4F,16#80,16#4F,16#C0,16#5F,16#C0,16#1F,16#40,16#10,16#40,16#10,16#40,16#10,16#40,16#10,16#C0,16#1F,16#C0,16#5F,16#80,16#4F,16#80,16#4F,16#00,16#00,16#00,16#00,16#00,16#00,16#00,16#00,	// 16#99
16#80,16#BF,16#80,16#BF,16#C0,16#BF,16#C0,16#BF,16#40,16#00,16#40,16#00,16#40,16#00,16#40,16#00,16#C0,16#BF,16#C0,16#BF,16#80,16#BF,16#80,16#BF,16#00,16#00,16#00,16#00,16#00,16#00,16#00,16#00,	// 16#9A
16#80,16#07,16#80,16#07,16#C0,16#0F,16#C0,16#0F,16#C0,16#09,16#40,16#0B,16#40,16#0E,16#40,16#0C,16#C0,16#0F,16#C0,16#07,16#80,16#07,16#80,16#07,16#00,16#00,16#00,16#00,16#00,16#00,16#00,16#00,	// 16#9B
16#C0,16#04,16#C0,16#04,16#C0,16#7F,16#C0,16#7F,16#40,16#FF,16#40,16#FF,16#40,16#84,16#40,16#84,16#40,16#84,16#40,16#84,16#40,16#C4,16#40,16#C4,16#40,16#40,16#40,16#40,16#00,16#00,16#00,16#00,	// 16#9C
16#00,16#1F,16#40,16#1F,16#C0,16#3F,16#80,16#3F,16#C0,16#71,16#C0,16#63,16#40,16#46,16#40,16#4C,16#C0,16#78,16#C0,16#71,16#80,16#3F,16#80,16#7F,16#00,16#5F,16#00,16#1F,16#00,16#00,16#00,16#00,	// 16#9D
16#40,16#08,16#C0,16#0C,16#C0,16#0C,16#80,16#04,16#80,16#07,16#00,16#03,16#00,16#03,16#00,16#03,16#80,16#07,16#80,16#04,16#C0,16#0C,16#C0,16#0C,16#40,16#08,16#00,16#00,16#00,16#00,16#00,16#00,	// 16#9E
16#80,16#00,16#80,16#00,16#C0,16#08,16#C0,16#08,16#40,16#08,16#40,16#08,16#C0,16#7F,16#C0,16#7F,16#80,16#FF,16#80,16#FF,16#00,16#88,16#00,16#88,16#00,16#C8,16#00,16#C8,16#00,16#40,16#00,16#40,	// 16#9F
16#80,16#01,16#80,16#01,16#C0,16#0B,16#C0,16#0B,16#40,16#2A,16#40,16#2A,16#40,16#6A,16#40,16#6A,16#C0,16#CF,16#80,16#CF,16#80,16#87,16#C0,16#87,16#40,16#00,16#40,16#00,16#00,16#00,16#00,16#00,	// 16#A0
16#00,16#00,16#00,16#00,16#40,16#08,16#40,16#08,16#40,16#28,16#40,16#28,16#C0,16#6F,16#C0,16#6F,16#C0,16#CF,16#C0,16#CF,16#40,16#80,16#40,16#80,16#40,16#00,16#40,16#00,16#00,16#00,16#00,16#00,	// 16#A1
16#80,16#07,16#80,16#07,16#C0,16#0F,16#C0,16#0F,16#40,16#28,16#40,16#28,16#40,16#68,16#40,16#68,16#C0,16#CF,16#C0,16#CF,16#80,16#87,16#80,16#87,16#00,16#00,16#00,16#00,16#00,16#00,16#00,16#00,	// 16#A2
16#80,16#0F,16#80,16#0F,16#C0,16#0F,16#C0,16#0F,16#40,16#20,16#40,16#20,16#40,16#60,16#40,16#60,16#C0,16#CF,16#80,16#CF,16#80,16#8F,16#C0,16#8F,16#40,16#00,16#40,16#00,16#00,16#00,16#00,16#00,	// 16#A3
16#C0,16#2F,16#C0,16#2F,16#C0,16#6F,16#C0,16#6F,16#00,16#48,16#00,16#48,16#00,16#68,16#00,16#68,16#C0,16#2F,16#C0,16#2F,16#C0,16#67,16#C0,16#67,16#00,16#40,16#00,16#40,16#00,16#00,16#00,16#00,	// 16#A4
16#C0,16#5F,16#C0,16#5F,16#C0,16#DF,16#C0,16#DF,16#00,16#8C,16#00,16#8C,16#00,16#C6,16#00,16#C6,16#00,16#43,16#00,16#43,16#C0,16#DF,16#C0,16#DF,16#C0,16#9F,16#C0,16#9F,16#00,16#00,16#00,16#00,	// 16#A5
16#00,16#32,16#00,16#32,16#00,16#7A,16#00,16#7A,16#00,16#4A,16#00,16#4A,16#00,16#4A,16#00,16#4A,16#00,16#7A,16#00,16#72,16#00,16#72,16#00,16#7A,16#00,16#0A,16#00,16#0A,16#00,16#00,16#00,16#00,	// 16#A6
16#00,16#32,16#00,16#32,16#00,16#7A,16#00,16#7A,16#00,16#4A,16#00,16#4A,16#00,16#4A,16#00,16#4A,16#00,16#7A,16#00,16#7A,16#00,16#32,16#00,16#32,16#00,16#02,16#00,16#02,16#00,16#00,16#00,16#00,	// 16#A7
16#80,16#03,16#80,16#03,16#C0,16#07,16#C0,16#07,16#40,16#6C,16#40,16#6C,16#40,16#68,16#40,16#68,16#C0,16#00,16#C0,16#00,16#80,16#00,16#80,16#00,16#00,16#00,16#00,16#00,16#00,16#00,16#00,16#00,	// 16#A8
16#00,16#1F,16#80,16#3F,16#C0,16#60,16#40,16#5F,16#40,16#5F,16#40,16#54,16#40,16#5E,16#40,16#5B,16#40,16#41,16#C0,16#60,16#80,16#3F,16#00,16#1F,16#00,16#00,16#00,16#00,16#00,16#00,16#00,16#00,	// 16#A9
16#00,16#04,16#00,16#04,16#00,16#04,16#00,16#04,16#00,16#04,16#00,16#04,16#00,16#04,16#00,16#04,16#80,16#07,16#80,16#07,16#80,16#07,16#80,16#07,16#00,16#00,16#00,16#00,16#00,16#00,16#00,16#00,	// 16#AA
16#80,16#21,16#80,16#21,16#00,16#7B,16#00,16#7B,16#00,16#7E,16#00,16#7E,16#20,16#0C,16#20,16#0D,16#60,16#1B,16#60,16#1A,16#E0,16#32,16#E0,16#32,16#A0,16#63,16#A0,16#63,16#20,16#01,16#20,16#01,	// 16#AB
16#80,16#21,16#80,16#21,16#00,16#7B,16#00,16#7B,16#C0,16#7E,16#C0,16#7E,16#C0,16#0D,16#C0,16#0D,16#40,16#1B,16#40,16#1B,16#40,16#36,16#40,16#36,16#E0,16#67,16#E0,16#67,16#E0,16#47,16#E0,16#47,	// 16#AC
16#00,16#00,16#00,16#00,16#80,16#03,16#80,16#03,16#C0,16#6F,16#C0,16#6F,16#C0,16#6F,16#C0,16#6F,16#80,16#03,16#80,16#03,16#00,16#00,16#00,16#00,16#00,16#00,16#00,16#00,16#00,16#00,16#00,16#00,	// 16#AD
16#00,16#03,16#00,16#03,16#80,16#07,16#80,16#07,16#C0,16#0C,16#C0,16#0C,16#40,16#08,16#40,16#08,16#00,16#03,16#00,16#03,16#80,16#07,16#80,16#07,16#C0,16#0C,16#C0,16#0C,16#40,16#08,16#40,16#08,	// 16#AE
16#40,16#08,16#40,16#08,16#C0,16#0C,16#C0,16#0C,16#80,16#07,16#80,16#07,16#00,16#03,16#00,16#03,16#40,16#08,16#40,16#08,16#C0,16#0C,16#C0,16#0C,16#80,16#07,16#80,16#07,16#00,16#03,16#00,16#03,	// 16#AF
16#20,16#49,16#20,16#49,16#90,16#24,16#90,16#24,16#40,16#92,16#40,16#92,16#20,16#49,16#20,16#49,16#90,16#24,16#90,16#24,16#40,16#92,16#40,16#92,16#20,16#49,16#20,16#49,16#90,16#24,16#90,16#24,	// 16#B0
16#50,16#55,16#50,16#55,16#A0,16#AA,16#A0,16#AA,16#50,16#55,16#50,16#55,16#A0,16#AA,16#A0,16#AA,16#50,16#55,16#50,16#55,16#A0,16#AA,16#A0,16#AA,16#50,16#55,16#50,16#55,16#A0,16#AA,16#A0,16#AA,	// 16#B1
16#B0,16#6D,16#B0,16#6D,16#60,16#DB,16#60,16#DB,16#D0,16#B6,16#D0,16#B6,16#B0,16#6D,16#B0,16#6D,16#60,16#DB,16#60,16#DB,16#D0,16#B6,16#D0,16#B6,16#B0,16#6D,16#B0,16#6D,16#60,16#DB,16#60,16#DB,	// 16#B2
16#00,16#00,16#00,16#00,16#00,16#00,16#00,16#00,16#00,16#00,16#00,16#00,16#F0,16#FF,16#F0,16#FF,16#F0,16#FF,16#F0,16#FF,16#00,16#00,16#00,16#00,16#00,16#00,16#00,16#00,16#00,16#00,16#00,16#00,	// 16#B3
16#00,16#00,16#00,16#00,16#00,16#04,16#00,16#04,16#00,16#04,16#00,16#04,16#F0,16#FF,16#F0,16#FF,16#F0,16#FF,16#F0,16#FF,16#00,16#00,16#00,16#00,16#00,16#00,16#00,16#00,16#00,16#00,16#00,16#00,	// 16#B4
16#C0,16#07,16#C0,16#0F,16#C0,16#0F,16#C0,16#1F,16#00,16#51,16#00,16#51,16#00,16#D1,16#00,16#D1,16#C0,16#9F,16#C0,16#8F,16#C0,16#0F,16#C0,16#07,16#00,16#00,16#00,16#00,16#00,16#00,16#00,16#00,	// 16#B5
16#C0,16#07,16#C0,16#0F,16#C0,16#4F,16#C0,16#5F,16#00,16#D1,16#00,16#91,16#00,16#91,16#00,16#D1,16#C0,16#5F,16#C0,16#4F,16#C0,16#0F,16#C0,16#07,16#00,16#00,16#00,16#00,16#00,16#00,16#00,16#00,	// 16#B6
16#C0,16#07,16#C0,16#0F,16#C0,16#8F,16#C0,16#9F,16#00,16#D1,16#00,16#D1,16#00,16#51,16#00,16#51,16#C0,16#1F,16#C0,16#0F,16#C0,16#0F,16#C0,16#07,16#00,16#00,16#00,16#00,16#00,16#00,16#00,16#00,	// 16#B7
16#00,16#1F,16#80,16#3F,16#C0,16#60,16#40,16#4E,16#40,16#5F,16#40,16#51,16#40,16#51,16#40,16#51,16#40,16#40,16#C0,16#60,16#80,16#3F,16#00,16#1F,16#00,16#00,16#00,16#00,16#00,16#00,16#00,16#00,	// 16#B8
16#00,16#09,16#00,16#09,16#F0,16#F9,16#F0,16#F9,16#F0,16#F9,16#F0,16#F9,16#00,16#00,16#00,16#00,16#00,16#00,16#00,16#00,16#F0,16#FF,16#F0,16#FF,16#F0,16#FF,16#F0,16#FF,16#00,16#00,16#00,16#00,	// 16#B9
16#00,16#00,16#00,16#00,16#F0,16#FF,16#F0,16#FF,16#F0,16#FF,16#F0,16#FF,16#00,16#00,16#00,16#00,16#00,16#00,16#00,16#00,16#F0,16#FF,16#F0,16#FF,16#F0,16#FF,16#F0,16#FF,16#00,16#00,16#00,16#00,	// 16#BA
16#00,16#09,16#00,16#09,16#F0,16#09,16#F0,16#09,16#F0,16#09,16#F0,16#09,16#00,16#08,16#00,16#08,16#00,16#08,16#00,16#08,16#F0,16#0F,16#F0,16#0F,16#F0,16#0F,16#F0,16#0F,16#00,16#00,16#00,16#00,	// 16#BB
16#00,16#09,16#00,16#09,16#00,16#F9,16#00,16#F9,16#00,16#F9,16#00,16#F9,16#00,16#01,16#00,16#01,16#00,16#01,16#00,16#01,16#00,16#FF,16#00,16#FF,16#00,16#FF,16#00,16#FF,16#00,16#00,16#00,16#00,	// 16#BC
16#00,16#04,16#00,16#04,16#00,16#FC,16#00,16#FC,16#00,16#FC,16#00,16#FC,16#00,16#04,16#00,16#04,16#00,16#04,16#00,16#04,16#00,16#FC,16#00,16#FC,16#00,16#FC,16#00,16#FC,16#00,16#00,16#00,16#00,	// 16#BD
16#00,16#0F,16#00,16#0F,16#80,16#1F,16#80,16#1F,16#E0,16#70,16#E0,16#70,16#E0,16#70,16#E0,16#70,16#80,16#19,16#80,16#19,16#00,16#09,16#00,16#09,16#00,16#00,16#00,16#00,16#00,16#00,16#00,16#00,	// 16#BE
16#00,16#F5,16#00,16#F5,16#00,16#FD,16#00,16#FD,16#C0,16#0F,16#C0,16#0F,16#C0,16#0F,16#C0,16#0F,16#00,16#FD,16#00,16#FD,16#00,16#F5,16#00,16#F5,16#00,16#00,16#00,16#00,16#00,16#00,16#00,16#00,	// 16#BF
16#00,16#00,16#00,16#00,16#00,16#00,16#00,16#00,16#00,16#00,16#00,16#00,16#00,16#FC,16#00,16#FC,16#00,16#FC,16#00,16#FC,16#00,16#04,16#00,16#04,16#00,16#04,16#00,16#04,16#00,16#04,16#00,16#04,	// 16#C0
16#00,16#04,16#00,16#04,16#00,16#04,16#00,16#04,16#00,16#04,16#00,16#04,16#00,16#FC,16#00,16#FC,16#00,16#FC,16#00,16#FC,16#00,16#04,16#00,16#04,16#00,16#04,16#00,16#04,16#00,16#04,16#00,16#04,	// 16#C1
16#00,16#04,16#00,16#04,16#00,16#04,16#00,16#04,16#00,16#04,16#00,16#04,16#F0,16#07,16#F0,16#07,16#F0,16#07,16#F0,16#07,16#00,16#04,16#00,16#04,16#00,16#04,16#00,16#04,16#00,16#04,16#00,16#04,	// 16#C2
16#00,16#00,16#00,16#00,16#00,16#00,16#00,16#00,16#00,16#00,16#00,16#00,16#F0,16#FF,16#F0,16#FF,16#F0,16#FF,16#F0,16#FF,16#00,16#04,16#00,16#04,16#00,16#04,16#00,16#04,16#00,16#04,16#00,16#04,	// 16#C3
16#00,16#04,16#00,16#04,16#00,16#04,16#00,16#04,16#00,16#04,16#00,16#04,16#00,16#04,16#00,16#04,16#00,16#04,16#00,16#04,16#00,16#04,16#00,16#04,16#00,16#04,16#00,16#04,16#00,16#04,16#00,16#04,	// 16#C4
16#00,16#04,16#00,16#04,16#00,16#04,16#00,16#04,16#00,16#04,16#00,16#04,16#F0,16#FF,16#F0,16#FF,16#F0,16#FF,16#F0,16#FF,16#00,16#04,16#00,16#04,16#00,16#04,16#00,16#04,16#00,16#04,16#00,16#04,	// 16#C5
16#80,16#21,16#80,16#21,16#C0,16#6B,16#C0,16#6B,16#40,16#4A,16#40,16#4A,16#40,16#6A,16#40,16#6A,16#C0,16#2F,16#80,16#2F,16#80,16#67,16#C0,16#67,16#40,16#40,16#40,16#40,16#00,16#00,16#00,16#00,	// 16#C6
16#C0,16#47,16#C0,16#4F,16#C0,16#CF,16#C0,16#DF,16#00,16#91,16#00,16#D1,16#00,16#D1,16#00,16#51,16#C0,16#DF,16#C0,16#CF,16#C0,16#8F,16#C0,16#87,16#00,16#00,16#00,16#00,16#00,16#00,16#00,16#00,	// 16#C7
16#00,16#00,16#00,16#00,16#00,16#FF,16#00,16#FF,16#00,16#FF,16#00,16#FF,16#00,16#01,16#00,16#01,16#00,16#01,16#00,16#01,16#00,16#F9,16#00,16#F9,16#00,16#F9,16#00,16#F9,16#00,16#09,16#00,16#09,	// 16#C8
16#00,16#00,16#00,16#00,16#F0,16#0F,16#F0,16#0F,16#F0,16#0F,16#F0,16#0F,16#00,16#08,16#00,16#08,16#00,16#08,16#00,16#08,16#F0,16#09,16#F0,16#09,16#F0,16#09,16#F0,16#09,16#00,16#09,16#00,16#09,	// 16#C9
16#00,16#09,16#00,16#09,16#00,16#F9,16#00,16#F9,16#00,16#F9,16#00,16#F9,16#00,16#01,16#00,16#01,16#00,16#01,16#00,16#01,16#00,16#F9,16#00,16#F9,16#00,16#F9,16#00,16#F9,16#00,16#09,16#00,16#09,	// 16#CA
16#00,16#09,16#00,16#09,16#F0,16#09,16#F0,16#09,16#F0,16#09,16#F0,16#09,16#00,16#08,16#00,16#08,16#00,16#08,16#00,16#08,16#F0,16#09,16#F0,16#09,16#F0,16#09,16#F0,16#09,16#00,16#09,16#00,16#09,	// 16#CB
16#00,16#00,16#00,16#00,16#F0,16#FF,16#F0,16#FF,16#F0,16#FF,16#F0,16#FF,16#00,16#00,16#00,16#00,16#00,16#00,16#00,16#00,16#F0,16#F9,16#F0,16#F9,16#F0,16#F9,16#F0,16#F9,16#00,16#09,16#00,16#09,	// 16#CC
16#00,16#09,16#00,16#09,16#00,16#09,16#00,16#09,16#00,16#09,16#00,16#09,16#00,16#09,16#00,16#09,16#00,16#09,16#00,16#09,16#00,16#09,16#00,16#09,16#00,16#09,16#00,16#09,16#00,16#09,16#00,16#09,	// 16#CD
16#00,16#09,16#00,16#09,16#F0,16#F9,16#F0,16#F9,16#F0,16#F9,16#F0,16#F9,16#00,16#00,16#00,16#00,16#00,16#00,16#00,16#00,16#F0,16#F9,16#F0,16#F9,16#F0,16#F9,16#F0,16#F9,16#00,16#09,16#00,16#09,	// 16#CE
16#40,16#20,16#C0,16#36,16#80,16#1F,16#80,16#19,16#80,16#19,16#80,16#19,16#80,16#19,16#80,16#19,16#80,16#19,16#80,16#19,16#80,16#1F,16#C0,16#36,16#40,16#20,16#00,16#00,16#00,16#00,16#00,16#00,	// 16#CF
16#00,16#00,16#00,16#03,16#80,16#A7,16#C0,16#AF,16#C0,16#AC,16#C0,16#CC,16#C0,16#6C,16#C0,16#EC,16#C0,16#BC,16#C0,16#BF,16#80,16#9F,16#00,16#0F,16#00,16#00,16#00,16#00,16#00,16#00,16#00,16#00,	// 16#D0
16#40,16#44,16#40,16#44,16#C0,16#7F,16#C0,16#7F,16#C0,16#7F,16#C0,16#7F,16#40,16#44,16#40,16#44,16#C0,16#60,16#C0,16#60,16#80,16#3F,16#80,16#3F,16#00,16#1F,16#00,16#1F,16#00,16#00,16#00,16#00,	// 16#D1
16#C0,16#1F,16#C0,16#1F,16#C0,16#5F,16#C0,16#5F,16#40,16#D2,16#40,16#92,16#40,16#92,16#40,16#D2,16#40,16#52,16#40,16#52,16#C0,16#18,16#C0,16#18,16#00,16#00,16#00,16#00,16#00,16#00,16#00,16#00,	// 16#D2
16#C0,16#DF,16#C0,16#DF,16#C0,16#DF,16#C0,16#1F,16#40,16#12,16#40,16#12,16#40,16#12,16#40,16#12,16#40,16#12,16#40,16#D2,16#C0,16#D8,16#C0,16#D8,16#00,16#00,16#00,16#00,16#00,16#00,16#00,16#00,	// 16#D3
16#C0,16#9F,16#C0,16#9F,16#C0,16#DF,16#C0,16#DF,16#40,16#72,16#40,16#72,16#40,16#32,16#40,16#32,16#40,16#12,16#40,16#12,16#C0,16#18,16#C0,16#18,16#00,16#00,16#00,16#00,16#00,16#00,16#00,16#00,	// 16#D4
16#00,16#42,16#00,16#42,16#00,16#7E,16#00,16#7E,16#00,16#7E,16#00,16#02,16#00,16#02,16#00,16#00,16#00,16#00,16#00,16#00,16#00,16#00,16#00,16#00,16#00,16#00,16#00,16#00,16#00,16#00,16#00,16#00,	// 16#D5
16#00,16#00,16#00,16#00,16#40,16#10,16#40,16#10,16#C0,16#5F,16#C0,16#5F,16#C0,16#DF,16#C0,16#DF,16#40,16#90,16#40,16#90,16#00,16#00,16#00,16#00,16#00,16#00,16#00,16#00,16#00,16#00,16#00,16#00,	// 16#D6
16#00,16#00,16#00,16#00,16#40,16#50,16#40,16#50,16#C0,16#DF,16#C0,16#9F,16#C0,16#9F,16#C0,16#DF,16#40,16#50,16#40,16#50,16#00,16#00,16#00,16#00,16#00,16#00,16#00,16#00,16#00,16#00,16#00,16#00,	// 16#D7
16#00,16#00,16#00,16#00,16#40,16#D0,16#40,16#D0,16#C0,16#DF,16#C0,16#1F,16#C0,16#1F,16#C0,16#DF,16#40,16#D0,16#40,16#D0,16#00,16#00,16#00,16#00,16#00,16#00,16#00,16#00,16#00,16#00,16#00,16#00,	// 16#D8
16#00,16#04,16#00,16#04,16#00,16#04,16#00,16#04,16#00,16#04,16#00,16#04,16#00,16#FC,16#00,16#FC,16#00,16#FC,16#00,16#FC,16#00,16#00,16#00,16#00,16#00,16#00,16#00,16#00,16#00,16#00,16#00,16#00,	// 16#D9
16#00,16#00,16#00,16#00,16#00,16#00,16#00,16#00,16#00,16#00,16#00,16#00,16#F0,16#07,16#F0,16#07,16#F0,16#07,16#F0,16#07,16#00,16#04,16#00,16#04,16#00,16#04,16#00,16#04,16#00,16#04,16#00,16#04,	// 16#DA
16#F0,16#FF,16#F0,16#FF,16#F0,16#FF,16#F0,16#FF,16#F0,16#FF,16#F0,16#FF,16#F0,16#FF,16#F0,16#FF,16#F0,16#FF,16#F0,16#FF,16#F0,16#FF,16#F0,16#FF,16#F0,16#FF,16#F0,16#FF,16#F0,16#FF,16#F0,16#FF,	// 16#DB
16#F0,16#03,16#F0,16#03,16#F0,16#03,16#F0,16#03,16#F0,16#03,16#F0,16#03,16#F0,16#03,16#F0,16#03,16#F0,16#03,16#F0,16#03,16#F0,16#03,16#F0,16#03,16#F0,16#03,16#F0,16#03,16#F0,16#03,16#F0,16#03,	// 16#DC
16#00,16#00,16#00,16#00,16#00,16#00,16#00,16#00,16#00,16#00,16#00,16#00,16#C0,16#7B,16#C0,16#7B,16#C0,16#7B,16#C0,16#7B,16#00,16#00,16#00,16#00,16#00,16#00,16#00,16#00,16#00,16#00,16#00,16#00,	// 16#DD
16#00,16#00,16#00,16#00,16#40,16#90,16#40,16#90,16#C0,16#DF,16#C0,16#DF,16#C0,16#5F,16#C0,16#5F,16#40,16#10,16#40,16#10,16#00,16#00,16#00,16#00,16#00,16#00,16#00,16#00,16#00,16#00,16#00,16#00,	// 16#DE
16#00,16#FC,16#00,16#FC,16#00,16#FC,16#00,16#FC,16#00,16#FC,16#00,16#FC,16#00,16#FC,16#00,16#FC,16#00,16#FC,16#00,16#FC,16#00,16#FC,16#00,16#FC,16#00,16#FC,16#00,16#FC,16#00,16#FC,16#00,16#FC,	// 16#DF
16#80,16#0F,16#80,16#0F,16#C0,16#1F,16#C0,16#1F,16#40,16#50,16#40,16#50,16#40,16#D0,16#40,16#D0,16#C0,16#9F,16#C0,16#9F,16#80,16#0F,16#80,16#0F,16#00,16#00,16#00,16#00,16#00,16#00,16#00,16#00,	// 16#E0
16#C0,16#3F,16#C0,16#3F,16#E0,16#7F,16#E0,16#7F,16#A0,16#40,16#A0,16#40,16#80,16#48,16#80,16#48,16#80,16#7F,16#80,16#7F,16#00,16#37,16#00,16#37,16#00,16#00,16#00,16#00,16#00,16#00,16#00,16#00,	// 16#E1
16#80,16#0F,16#80,16#0F,16#C0,16#5F,16#C0,16#5F,16#40,16#D0,16#40,16#90,16#40,16#90,16#40,16#D0,16#C0,16#5F,16#C0,16#5F,16#80,16#0F,16#80,16#0F,16#00,16#00,16#00,16#00,16#00,16#00,16#00,16#00,	// 16#E2
16#80,16#0F,16#80,16#0F,16#C0,16#1F,16#C0,16#9F,16#40,16#90,16#40,16#D0,16#40,16#D0,16#40,16#50,16#40,16#50,16#C0,16#1F,16#C0,16#1F,16#80,16#0F,16#80,16#0F,16#00,16#00,16#00,16#00,16#00,16#00,	// 16#E3
16#80,16#27,16#80,16#27,16#C0,16#6F,16#C0,16#6F,16#40,16#48,16#40,16#68,16#40,16#68,16#40,16#28,16#C0,16#6F,16#C0,16#6F,16#80,16#47,16#80,16#47,16#00,16#00,16#00,16#00,16#00,16#00,16#00,16#00,	// 16#E4
16#80,16#4F,16#80,16#4F,16#C0,16#DF,16#C0,16#DF,16#40,16#90,16#40,16#90,16#40,16#D0,16#40,16#50,16#C0,16#5F,16#C0,16#DF,16#80,16#CF,16#80,16#8F,16#00,16#80,16#00,16#00,16#00,16#00,16#00,16#00,	// 16#E5
16#10,16#00,16#10,16#00,16#F0,16#0F,16#F0,16#0F,16#E0,16#0F,16#E0,16#0F,16#40,16#00,16#40,16#00,16#40,16#00,16#40,16#00,16#C0,16#0F,16#80,16#0F,16#80,16#0F,16#C0,16#0F,16#40,16#00,16#40,16#00,	// 16#E6
16#40,16#20,16#C0,16#3F,16#C0,16#3F,16#C0,16#3F,16#40,16#1B,16#00,16#1B,16#00,16#1B,16#00,16#1B,16#00,16#1B,16#00,16#1F,16#00,16#0E,16#00,16#00,16#00,16#00,16#00,16#00,16#00,16#00,16#00,16#00,	// 16#E7
16#40,16#40,16#C0,16#7F,16#C0,16#7F,16#C0,16#7F,16#C0,16#7F,16#40,16#5B,16#40,16#1B,16#00,16#1B,16#00,16#1B,16#00,16#1B,16#00,16#1B,16#00,16#1F,16#00,16#0E,16#00,16#00,16#00,16#00,16#00,16#00,	// 16#E8
16#80,16#1F,16#80,16#1F,16#C0,16#1F,16#C0,16#1F,16#40,16#40,16#40,16#40,16#40,16#C0,16#40,16#C0,16#C0,16#9F,16#C0,16#9F,16#80,16#1F,16#80,16#1F,16#00,16#00,16#00,16#00,16#00,16#00,16#00,16#00,	// 16#E9
16#80,16#1F,16#80,16#1F,16#C0,16#5F,16#C0,16#5F,16#40,16#C0,16#40,16#80,16#40,16#80,16#40,16#C0,16#C0,16#5F,16#C0,16#5F,16#80,16#1F,16#80,16#1F,16#00,16#00,16#00,16#00,16#00,16#00,16#00,16#00,	// 16#EA
16#80,16#1F,16#80,16#1F,16#C0,16#9F,16#C0,16#9F,16#40,16#C0,16#40,16#C0,16#40,16#40,16#40,16#40,16#C0,16#1F,16#C0,16#1F,16#80,16#1F,16#80,16#1F,16#00,16#00,16#00,16#00,16#00,16#00,16#00,16#00,	// 16#EB
16#10,16#00,16#10,16#00,16#10,16#0F,16#10,16#0F,16#90,16#0F,16#90,16#0F,16#B0,16#20,16#B0,16#20,16#E0,16#60,16#E0,16#60,16#C0,16#CF,16#C0,16#CF,16#00,16#8F,16#00,16#8F,16#00,16#00,16#00,16#00,	// 16#EC
16#00,16#1C,16#00,16#1C,16#40,16#1E,16#40,16#1E,16#C0,16#47,16#C0,16#47,16#C0,16#C7,16#C0,16#C7,16#40,16#9E,16#40,16#9E,16#00,16#1C,16#00,16#1C,16#00,16#00,16#00,16#00,16#00,16#00,16#00,16#00,	// 16#ED
16#00,16#C0,16#00,16#C0,16#00,16#C0,16#00,16#C0,16#00,16#C0,16#00,16#C0,16#00,16#C0,16#00,16#C0,16#00,16#C0,16#00,16#C0,16#00,16#C0,16#00,16#C0,16#00,16#C0,16#00,16#00,16#00,16#00,16#00,16#00,	// 16#EE
16#00,16#00,16#00,16#00,16#00,16#00,16#00,16#00,16#00,16#20,16#00,16#20,16#00,16#60,16#00,16#60,16#00,16#C0,16#00,16#C0,16#00,16#80,16#00,16#80,16#00,16#00,16#00,16#00,16#00,16#00,16#00,16#00,	// 16#EF
16#00,16#06,16#00,16#06,16#00,16#06,16#00,16#06,16#00,16#06,16#00,16#06,16#00,16#06,16#00,16#06,16#00,16#06,16#00,16#06,16#00,16#06,16#00,16#06,16#00,16#00,16#00,16#00,16#00,16#00,16#00,16#00,	// 16#F0
16#80,16#08,16#80,16#08,16#80,16#08,16#80,16#08,16#80,16#3E,16#80,16#3E,16#80,16#3E,16#80,16#3E,16#80,16#08,16#80,16#08,16#80,16#08,16#80,16#08,16#00,16#00,16#00,16#00,16#00,16#00,16#00,16#00,	// 16#F1
16#80,16#04,16#80,16#04,16#80,16#04,16#80,16#04,16#80,16#04,16#80,16#04,16#80,16#04,16#80,16#04,16#80,16#04,16#80,16#04,16#80,16#04,16#80,16#04,16#00,16#00,16#00,16#00,16#00,16#00,16#00,16#00,	// 16#F2
16#80,16#88,16#80,16#A9,16#00,16#A9,16#00,16#AB,16#00,16#FA,16#C0,16#DE,16#C0,16#0D,16#C0,16#0D,16#40,16#1B,16#40,16#1B,16#40,16#36,16#40,16#36,16#E0,16#67,16#E0,16#67,16#E0,16#07,16#E0,16#07,	// 16#F3
16#00,16#38,16#00,16#38,16#00,16#7C,16#00,16#7C,16#00,16#44,16#00,16#44,16#C0,16#7F,16#C0,16#7F,16#C0,16#7F,16#C0,16#7F,16#00,16#40,16#00,16#40,16#C0,16#7F,16#C0,16#7F,16#C0,16#7F,16#C0,16#7F,	// 16#F4
16#40,16#00,16#40,16#00,16#60,16#26,16#60,16#36,16#20,16#7F,16#20,16#7F,16#20,16#59,16#20,16#49,16#20,16#49,16#A0,16#49,16#E0,16#4F,16#E0,16#4F,16#C0,16#66,16#40,16#66,16#00,16#20,16#00,16#20,	// 16#F5
16#00,16#04,16#00,16#04,16#00,16#04,16#00,16#04,16#80,16#35,16#80,16#35,16#80,16#35,16#80,16#35,16#00,16#04,16#00,16#04,16#00,16#04,16#00,16#04,16#00,16#00,16#00,16#00,16#00,16#00,16#00,16#00,	// 16#F6
16#00,16#00,16#10,16#00,16#10,16#00,16#10,16#00,16#30,16#00,16#30,16#00,16#30,16#00,16#20,16#00,16#00,16#00,16#00,16#00,16#00,16#00,16#00,16#00,16#00,16#00,16#00,16#00,16#00,16#00,16#00,16#00,	// 16#F7
16#00,16#00,16#00,16#00,16#00,16#38,16#00,16#38,16#00,16#7C,16#00,16#7C,16#00,16#44,16#00,16#44,16#00,16#44,16#00,16#44,16#00,16#7C,16#00,16#7C,16#00,16#38,16#00,16#38,16#00,16#00,16#00,16#00,	// 16#F8
16#00,16#60,16#00,16#60,16#00,16#60,16#00,16#00,16#00,16#00,16#00,16#00,16#00,16#00,16#00,16#00,16#00,16#00,16#00,16#60,16#00,16#60,16#00,16#60,16#00,16#00,16#00,16#00,16#00,16#00,16#00,16#00,	// 16#F9
16#00,16#00,16#00,16#00,16#00,16#00,16#00,16#00,16#00,16#00,16#00,16#00,16#00,16#06,16#00,16#06,16#00,16#06,16#00,16#00,16#00,16#00,16#00,16#00,16#00,16#00,16#00,16#00,16#00,16#00,16#00,16#00,	// 16#FA
16#00,16#00,16#00,16#00,16#00,16#00,16#00,16#20,16#00,16#24,16#00,16#64,16#00,16#7C,16#00,16#7C,16#00,16#7C,16#00,16#04,16#00,16#04,16#00,16#00,16#00,16#00,16#00,16#00,16#00,16#00,16#00,16#00,	// 16#FB
16#00,16#00,16#00,16#00,16#00,16#44,16#00,16#54,16#00,16#54,16#00,16#54,16#00,16#7C,16#00,16#7C,16#00,16#7C,16#00,16#28,16#00,16#00,16#00,16#00,16#00,16#00,16#00,16#00,16#00,16#00,16#00,16#00,	// 16#FC
16#00,16#00,16#00,16#00,16#00,16#44,16#00,16#44,16#00,16#4C,16#00,16#4C,16#00,16#5C,16#00,16#5C,16#00,16#74,16#00,16#74,16#00,16#24,16#00,16#24,16#00,16#00,16#00,16#00,16#00,16#00,16#00,16#00,	// 16#FD
16#00,16#00,16#00,16#00,16#00,16#00,16#00,16#00,16#C0,16#3F,16#C0,16#3F,16#C0,16#3F,16#C0,16#3F,16#C0,16#3F,16#C0,16#3F,16#C0,16#3F,16#C0,16#3F,16#00,16#00,16#00,16#00,16#00,16#00,16#00,16#00,	// 16#FE
16#00,16#00,16#00,16#00,16#00,16#00,16#00,16#00,16#00,16#00,16#00,16#00,16#00,16#00,16#00,16#00,16#00,16#00,16#00,16#00,16#00,16#00,16#00,16#00,16#00,16#00,16#00,16#00,16#00,16#00,16#00,16#00 	// 16#FF
];



